(* PLC project Unnamed, Unknown Unnamed 1 *)
(* stored: creationDateTime 2024-09-14T19:27:39, modificationDateTime 2024-09-14T19:56:38 *)

PROGRAM counter
  VAR
    input_register AT %IW0.0 : INT;
    output_register AT %QW0.0 : INT;
  END_VAR

            output_register := input_register;
          
END_PROGRAM

CONFIGURATION Config0
  RESOURCE Res0 ON PLC
    TASK task0(INTERVAL := T#20ms, PRIORITY := 0);
    PROGRAM instance0 WITH task0 : counter;
  END_RESOURCE
END_CONFIGURATION
